// TIA Portal V16 export
// export: Created 2025-05-30T16:36:21.7686834Z, ExportSetting WithDefaults, DisplayName Totally Integrated Automation Portal, DisplayVersion V16, DisplayName TIA Portal Version Control Interface, DisplayVersion V16, DisplayName TIA Portal Openness, DisplayVersion V16, DisplayName STEP 7 Professional, DisplayVersion V16, DisplayName STEP 7 Safety, DisplayVersion V16, DisplayName WinCC Advanced, DisplayVersion V16
DATA_BLOCK "DriveConfirmation_Function_Axis 5"   // DB49
VERSION : 0.1
// stored: AutoNumber true, InstanceOfName DriveConfirmation_Function, InstanceOfType FB
"DriveConfirmation_Function"
   // VAR_INPUT
   //    "System RUN" : Bool;
   //    "Drive Ouput Q" : Bool;
   //    "Drive Ready Signal" : Bool;
   //    DelayTime : Time;
   // END_VAR
   // VAR_OUTPUT
   //    "Timer ET" : Time;
   //    "Ouput WORD" : Bool;
   // END_VAR
BEGIN
END_DATA_BLOCK
